SYSTEM DRILL_VIEWL (* Drill System View + HMI *)
  (* Standard: 61499-1; Classification: Simulation; ApplicationDomain: Transfer Lines; Function: Drillingd *)
  (* Version 0.1, 2004-10-18, JHC, Rockwell Automation, Changed loader/unloader to SOL_VIEWL. *)
  (* Version 0.0, 2002-04-25, JHC, Rockwell Automation, Adapted from TESTBED_VIEWL *)
  DEVICE HMI : FRAME_DEVICE(BOUNDS := [100,100,375,200], GRID := [1,1])
    RESOURCE RES1 : PANEL_RESOURCE
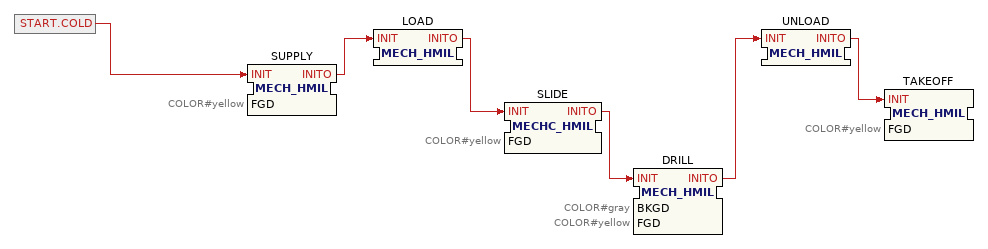
      FBS
        SUPPLY : MECH_HMIL(FGD := COLOR#yellow);
        LOAD : MECH_HMIL;
        DRILL : MECH_HMIL(BKGD := COLOR#gray, FGD := COLOR#yellow);
        SLIDE : MECHC_HMIL(FGD := COLOR#yellow);
        UNLOAD : MECH_HMIL;
        TAKEOFF : MECH_HMIL(FGD := COLOR#yellow);
      END_FBS
      EVENT_CONNECTIONS
        START.COLD TO SUPPLY.INIT;
        SUPPLY.INITO TO LOAD.INIT;
        LOAD.INITO TO SLIDE.INIT;
        SLIDE.INITO TO DRILL.INIT;
        DRILL.INITO TO UNLOAD.INIT;
        UNLOAD.INITO TO TAKEOFF.INIT;
      END_CONNECTIONS
    END_RESOURCE
  END_DEVICE
  DEVICE VIEW : FRAME_DEVICE(BOUNDS := [475,100,220,300])
    RESOURCE INPUT : VIEW_PANEL(DIA := 25, SIZE := [6,5], VERTICAL := 1)
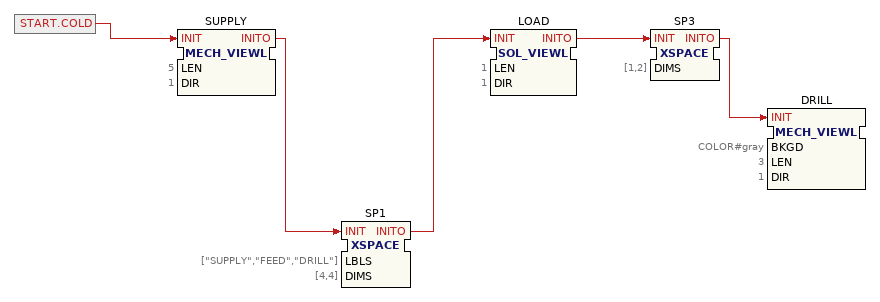
      FBS
        SUPPLY : MECH_VIEWL(LEN := 5, DIR := 1); (* Supply transfer mechanism *)
        SP1 : XSPACE(LBLS := ["SUPPLY","FEED","DRILL"], DIMS := [4,4]);
        LOAD : SOL_VIEWL(LEN := 1, DIR := 1); (* Loader mechanism *)
        SP3 : XSPACE(DIMS := [1,2]);
        DRILL : MECH_VIEWL(BKGD := COLOR#gray, LEN := 3, DIR := 1);
      END_FBS
      EVENT_CONNECTIONS
        START.COLD TO SUPPLY.INIT;
        SUPPLY.INITO TO SP1.INIT;
        SP1.INITO TO LOAD.INIT;
        LOAD.INITO TO SP3.INIT;
        SP3.INITO TO DRILL.INIT;
      END_CONNECTIONS
    END_RESOURCE
    RESOURCE OUTPUT : VIEW_PANEL(DIA := 25, SIZE := [6,5])
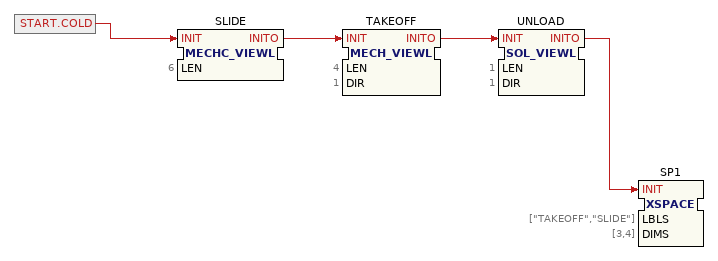
      FBS
        SLIDE : MECHC_VIEWL(LEN := 6);
        TAKEOFF : MECH_VIEWL(LEN := 4, DIR := 1); (* Takeoff Transfer *)
        UNLOAD : SOL_VIEWL(LEN := 1, DIR := 1); (* Unloader Mechanism *)
        SP1 : XSPACE(LBLS := ["TAKEOFF","SLIDE"], DIMS := [3,4]);
      END_FBS
      EVENT_CONNECTIONS
        START.COLD TO SLIDE.INIT;
        SLIDE.INITO TO TAKEOFF.INIT;
        TAKEOFF.INITO TO UNLOAD.INIT;
        UNLOAD.INITO TO SP1.INIT;
      END_CONNECTIONS
    END_RESOURCE
  END_DEVICE
END_SYSTEM
